DATA_BLOCK "mqttGlobals"
TITLE = 'MQTT CONSTANTS'
{ S7_Optimized_Access := 'FALSE' }
AUTHOR : Brand
VERSION : 0.1
NON_RETAIN
   STRUCT
      MQTT_KEEPALIVE : Time;
      MQTT_SOCKET_TIMEOUT : Time;
      TCP_RECVBUFFERSIZE : Int;   // size of TCP receive buffer
      TCP_MAXRECVSIZE : Int;   // TCP max receive packet size
      TCP_SENDBUFFERSIZE : Int;
      TCP_TIMEOUT : Time;   // timeout value for TCP connection MQtt States
      MQTT_STATE_DISCONNECT : Int;
      MQTT_STATE_DISCONNECTING : Int;
      MQTT_CONNECTION_TIMEOUT : Int;
      MQTT_CONNECTION_LOST : Int;
      MQTT_CONNECT_FAILED : Int;
      MQTT_DISCONNECTED : Int;
      MQTT_CONNECTING : Int;
      MQTT_CONNECTED : Int;
      MQTT_CONN_ACCEPTED : Int;
      MQTT_CONN_BAD_PROTOCOL : Int;
      MQTT_CONN_BAD_CLIENT_ID : Int;
      MQTT_CONN_SRVUNAVAIL : Int;
      MQTT_CONN_BAD_CREDEN : Int;
      MQTT_CONN_UNAUTHORIZED : Int;   // Packet headers
      MQTTCONNECT : Int;
      MQTTCONNACK : Int;
      MQTTPUBLISH : Int;
      MQTTPUBACK : Int;
      MQTTPUBREC : Int;
      MQTTPUBREL : Int;
      MQTTPUBCOMP : Int;
      MQTTSUBSCRIBE : Int;
      MQTTSUBACK : Int;
      MQTTUNSUBSCRIBE : Int;
      MQTTUNSUBACK : Int;
      MQTTPINGREQ : Int;
      MQTTPINGRESP : Int;
      MQTTDISCONNECT : Int;
      MQTTReserved : Int;
      MQTTQOS0 : Int;
      MQTTQOS1 : Int;
      MQTTQOS2 : Int;
   END_STRUCT;


BEGIN
   MQTT_KEEPALIVE := T#15S;
   MQTT_SOCKET_TIMEOUT := T#15S;
   TCP_RECVBUFFERSIZE := 8192;
   TCP_MAXRECVSIZE := 4096;
   TCP_SENDBUFFERSIZE := 4096;
   TCP_TIMEOUT := T#30S;
   MQTT_STATE_DISCONNECT := -6;
   MQTT_STATE_DISCONNECTING := -5;
   MQTT_CONNECTION_TIMEOUT := -4;
   MQTT_CONNECTION_LOST := -3;
   MQTT_CONNECT_FAILED := -2;
   MQTT_DISCONNECTED := -1;
   MQTT_CONNECTING := 0;
   MQTT_CONNECTED := 1;
   MQTT_CONN_ACCEPTED := 0;
   MQTT_CONN_BAD_PROTOCOL := 1;
   MQTT_CONN_BAD_CLIENT_ID := 2;
   MQTT_CONN_SRVUNAVAIL := 3;
   MQTT_CONN_BAD_CREDEN := 4;
   MQTT_CONN_UNAUTHORIZED := 5;
   MQTTCONNECT := 16;
   MQTTCONNACK := 32;
   MQTTPUBLISH := 48;
   MQTTPUBACK := 64;
   MQTTPUBREC := 80;
   MQTTPUBREL := 96;
   MQTTPUBCOMP := 112;
   MQTTSUBSCRIBE := 130;
   MQTTSUBACK := 144;
   MQTTUNSUBSCRIBE := 160;
   MQTTUNSUBACK := 176;
   MQTTPINGREQ := 192;
   MQTTPINGRESP := 208;
   MQTTDISCONNECT := 224;
   MQTTReserved := 240;
   MQTTQOS0 := 0;
   MQTTQOS1 := 1;
   MQTTQOS2 := 2;

END_DATA_BLOCK

